FUNCTION_BLOCK FB_Joystick
VAR_INPUT
	bEnable : BOOL;
	fNormalizedInput : LREAL;
	stParam : ST_Parameters;
END_VAR
VAR_OUTPUT
	fOuput : LREAL;
END_VAR
VAR
END_VAR

IF bEnable THEN
	fOuput := fNormalizedInput*Parameters.stParam.fMaxVelocityLimit;
ELSE
	fOuput := 0.0;
END_IF

END_FUNCTION_BLOCK

(* stored: Version 1.1.0.1, ProductVersion 3.1.4024.10
   POU FB_Joystick: Id {c7d518e7-72f7-41d3-8eec-d60f2a61bb42}, SpecialFunc None *)
